{attribute 'qualified_only'}
VAR_GLOBAL
	EmTeste:BOOL;
	LinhaSelecionada:INT;
	TesteHora:DATE;
	Teste2:DT;
END_VAR

(* stored: Version 1.1.0.1, ProductVersion 3.1.4024.13
   GVL Testes: Id {e31e838f-a1ca-43c0-ab66-af312cdf88da} *)
